FUNCTION_BLOCK SystemTime
VAR_INPUT
END_VAR
VAR_OUTPUT
END_VAR
VAR
END_VAR


fbGetLocalSystemTime(
	sNetID:= , 
	bEnable:= TRUE, 
	dwCycle:= 1, 
	dwOpt:= , 
	tTimeout:= , 
	bValid=> , 
	systemTime=> , 
	tzID=> );

Lib.GVL_DECI.sSystemDateTime :=  SYSTEMTIME_TO_STRING(Lib.GVL_DECI.fbGetLocalSystemTime.systemTime);
Lib.GVL_DECI.sSystemDate:= MID(STR:=Lib.GVL_DECI.sSystemDateTime, LEN:=10, POS:=1);
Lib.GVL_DECI.sSystemTime:= MID(STR:=Lib.GVL_DECI.sSystemDateTime, LEN:=8, POS:=12);

END_FUNCTION_BLOCK

(* stored: Version 1.1.0.1, ProductVersion 3.1.4024.12
   POU SystemTime: Id {044d0b00-502d-4d11-b206-5a75c97f8b00}, SpecialFunc None *)
